Yaskawa INFORM job: R1_W68-69(-90,-90)KM-OK-R2.JBI

/JOB
//NAME R1_W68-69(-90,-90)KM-OK-R2
///FOLDERNAME KRIS-SCIANA
//POS
///NPOS 37,37,0,3,0,0
///TOOL 0
///POSTYPE PULSE
///PULSE
C00000=-71699,4137,-33042,5531,91540,-26236
C00001=-120734,60189,59157,-4507,90133,53626
C00002=-120735,60186,59153,-4507,90134,53626
C00003=-121416,57763,57239,-4573,90029,53399
C00004=-121416,58241,58485,-4573,89510,53419
C00005=-121416,57763,57239,-4573,90029,53399
C00006=-121422,54955,54240,-4576,90430,53382
C00007=-121416,57763,57239,-4573,90029,53399
C00008=-111745,64559,70342,-20824,88560,57952
C00009=-112562,64120,69824,-20938,88442,57682
C00010=-111745,64559,70342,-20824,88560,57952
C00011=-120735,60233,59207,1568,97150,55574
C00012=-120734,60240,59215,1568,97148,55574
C00013=-120752,52948,31898,-27650,99286,-23836
C00014=-120734,59915,58842,2152,77537,-66258
C00015=-120734,59888,58811,2152,77542,-66258
C00016=-121262,57513,57182,2191,77339,-66443
C00017=-121262,57971,58365,2192,76844,-66452
C00018=-121262,57513,57182,2191,77339,-66443
C00019=-121266,55611,55232,2174,77564,-66440
C00020=-121262,57513,57182,2191,77339,-66443
C00021=-118819,57495,56763,2012,77525,-65597
C00022=-118206,57747,57314,1968,77300,-65390
C00023=-118819,57495,56763,2012,77525,-65597
C00024=-120734,59810,58720,-4331,84296,-67542
C00025=-120734,59832,58746,-4331,84292,-67542
C00026=-112141,52965,27873,23391,110918,28823
C00027=-106926,60351,59343,37595,103591,82494
C00028=-106926,60328,59317,37596,103595,82495
C00029=-83178,34766,16067,-1688,101215,86979
C00030=-107060,63407,62879,37458,103163,82282
C00031=-107025,61867,60184,37617,103844,82542
C00032=-112724,8742,-7432,-9788,101180,76515
C00033=-111971,9216,-5538,-16274,100907,76551
C00034=-109253,13785,-6794,-16748,105993,76804
C00035=-109220,18531,-23148,-18491,117951,74934
C00036=6001,25874,-16138,-19603,78346,75518
BC00000=45279,739780,873899
BC00001=88189,688652,601070
BC00002=84996,686395,577743
BC00003=83719,685493,568412
BC00004=83719,685493,568412
BC00005=83719,685493,568412
BC00006=83719,685493,568412
BC00007=83719,685493,568412
BC00008=83719,685493,568412
BC00009=83719,685493,568412
BC00010=83719,685493,568412
BC00011=72457,696409,570741
BC00012=74794,699714,593690
BC00013=162028,676418,516181
BC00014=156585,666650,613979
BC00015=158547,664946,588616
BC00016=159332,664264,578471
BC00017=159332,664264,578471
BC00018=159332,664264,578471
BC00019=159332,664264,578468
BC00020=159332,664264,578471
BC00021=159332,664264,578471
BC00022=159332,664264,578471
BC00023=159332,664264,578471
BC00024=177049,680818,585957
BC00025=176054,683477,610953
BC00026=109653,713304,532565
BC00027=69562,731313,485236
BC00028=72376,725585,470052
BC00029=73330,723643,464903
BC00030=73501,723294,463979
BC00031=73501,723294,463979
BC00032=73330,723643,464904
BC00033=73330,723643,464904
BC00034=73330,723643,464904
BC00035=73330,723644,464900
BC00036=73330,723644,757340
///POSTYPE BASE
///RECTAN
///RCONF 0,0,0,0,0,0,0,0,0,0,0,0,0,0,0,0,0,0,0,0,0,0,0,0
P00006=0.222,-3.123,-1.508,0.0000,0.0000,0.0000
P00021=-0.225,-6.128,-0.405,0.0000,0.0000,0.0000
P00022=0.222,-3.123,-1.508,0.0000,0.0000,0.0000
//INST
///DATE 2024/07/23 16:22
///ATTR SC,RW
///GROUP1 RB1,BS1
NOP
SFTOF
MOVJ C00000 BC00000 VJ=100.00
MOVJ C00001 BC00001 VJ=100.00
MOVL C00002 BC00002 V=100.0
MOVL C00003 BC00003 V=60.0
REFP 3 C00004 BC00004
CALL JOB:SEARCH-R1
SET P021 P006
SFTON P021
MOVL C00005 BC00005 V=60.0
REFP 3 C00006 BC00006
CALL JOB:SEARCH-R1
SET P021 P006
SFTON P021
MOVL C00007 BC00007 V=60.0
MOVL C00008 BC00008 V=60.0
REFP 3 C00009 BC00009
CALL JOB:SEARCH-R1
SET P021 P006
SFTON P021
MOVL C00010 BC00010 V=60.0
MOVL C00011 BC00011 V=100.0
MOVL C00012 BC00012 V=166.7
'Path VIA1138
SFTOF
MOVJ C00013 BC00013 VJ=100.00
'Path S759 (for W102)
SFTOF
MOVJ C00014 BC00014 VJ=100.00
MOVL C00015 BC00015 V=100.0
MOVL C00016 BC00016 V=60.0
REFP 3 C00017 BC00017
CALL JOB:SEARCH-R1
SET P022 P006
SFTON P022
MOVL C00018 BC00018 V=60.0
REFP 3 C00019 BC00019
CALL JOB:SEARCH-R1
SET P022 P006
SFTON P022
MOVL C00020 BC00020 V=60.0
MOVL C00021 BC00021 V=60.0
REFP 3 C00022 BC00022
CALL JOB:SEARCH-R1
SET P022 P006
SFTON P022
MOVL C00023 BC00023 V=60.0
MOVL C00024 BC00024 V=166.7
MOVL C00025 BC00025 V=166.7
'Path VIA1139
SFTOF
MOVJ C00026 BC00026 VJ=100.00
'Path W102
SFTOF
SFTON P022
MOVJ C00027 BC00027 VJ=100.00
MOVL C00028 BC00028 V=333.3
MOVL C00029 BC00029 V=166.7 PL=0
REFP 1 C00030 BC00030
REFP 2 C00031 BC00031
MACRO1 MJ#(0) ARGF9
ARCON
SFTON P021
MOVL C00032 BC00032 V=10.8
MOVL C00033 BC00033 V=10.8
ARCOF
MOVL C00034 BC00034 V=166.7
SFTOF
MOVJ C00035 BC00035 VJ=100.00
MOVJ C00036 BC00036 VJ=100.00
END
